// TIA Portal V18 export
// export: Created 2026-06-22T15:41:34.752897Z, ExportSetting WithDefaults, DisplayName Totally Integrated Automation Portal, DisplayVersion V18, DisplayName TIA Portal Openness, DisplayVersion V18, DisplayName TIA Portal Version Control Interface, DisplayVersion V18, DisplayName STEP 7 Professional, DisplayVersion V18, DisplayName STEP 7 Safety, DisplayVersion V18, DisplayName WinCC Professional, DisplayVersion V18
ORGANIZATION_BLOCK "OB30_Encoder_100ms"   // OB30, LAD, CyclicInterrupt
{ S7_Optimized_Access := 'TRUE' }
VERSION : 0.1
// stored: AutoNumber true, IsIECCheckEnabled false, SetENOAutomatically false
   VAR_INPUT
      Initial_Call : Bool;   // Initial call of this OB
      Event_Count : Int;   // Events discarded
   END_VAR
BEGIN

REGION Network 1: Đọc giá trị HSC và tính Delta Count
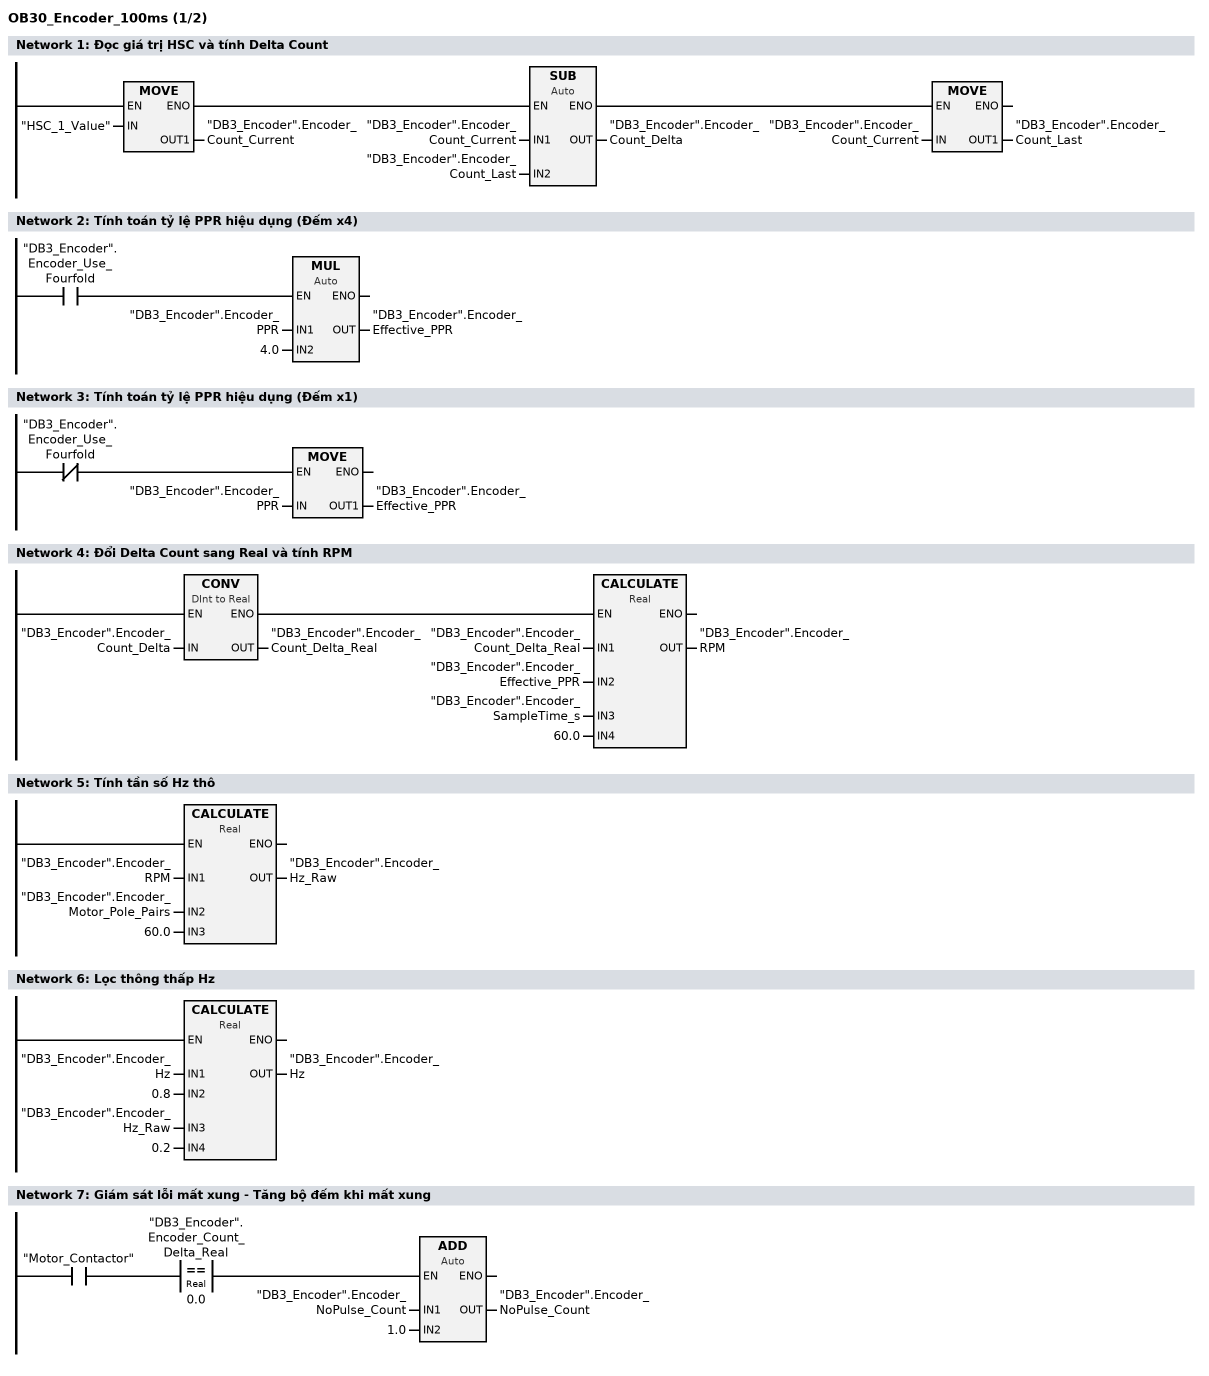
   RUNG wire#powerrail
      { S7_GenerateENO := "TRUE" } Move(in := "HSC_1_Value", out1 => "DB3_Encoder".Encoder_Count_Current)
      { S7_GenerateENO := "TRUE" } Sub(in1 := "DB3_Encoder".Encoder_Count_Current, in2 := "DB3_Encoder".Encoder_Count_Last, out => "DB3_Encoder".Encoder_Count_Delta)
      { S7_GenerateENO := "TRUE" } Move(in := "DB3_Encoder".Encoder_Count_Current, out1 => "DB3_Encoder".Encoder_Count_Last)
   END_RUNG
   // the same network as SCL:
   // ENO of a box is taken as its EN; it also drops when the box reports an error
   "DB3_Encoder".Encoder_Count_Current := "HSC_1_Value";
   "DB3_Encoder".Encoder_Count_Delta := "DB3_Encoder".Encoder_Count_Current - "DB3_Encoder".Encoder_Count_Last;
   "DB3_Encoder".Encoder_Count_Last := "DB3_Encoder".Encoder_Count_Current;
END_REGION

REGION Network 2: Tính toán tỷ lệ PPR hiệu dụng (Đếm x4)
   RUNG wire#powerrail
      Contact( "DB3_Encoder".Encoder_Use_Fourfold )
      { S7_GenerateENO := "TRUE" } Mul(in1 := "DB3_Encoder".Encoder_PPR, in2 := 4.0, out => "DB3_Encoder".Encoder_Effective_PPR)
   END_RUNG
   // the same network as SCL:
   IF "DB3_Encoder".Encoder_Use_Fourfold THEN
       "DB3_Encoder".Encoder_Effective_PPR := "DB3_Encoder".Encoder_PPR * 4.0;
   END_IF;
END_REGION

REGION Network 3: Tính toán tỷ lệ PPR hiệu dụng (Đếm x1)
   RUNG wire#powerrail
      I_Contact( "DB3_Encoder".Encoder_Use_Fourfold )
      { S7_GenerateENO := "TRUE" } Move(in := "DB3_Encoder".Encoder_PPR, out1 => "DB3_Encoder".Encoder_Effective_PPR)
   END_RUNG
   // the same network as SCL:
   IF NOT "DB3_Encoder".Encoder_Use_Fourfold THEN
       "DB3_Encoder".Encoder_Effective_PPR := "DB3_Encoder".Encoder_PPR;
   END_IF;
END_REGION

REGION Network 4: Đổi Delta Count sang Real và tính RPM
   RUNG wire#powerrail
      { S7_Templates := "[SrcType := DInt, DestType := Real]"; S7_GenerateENO := "TRUE" } Convert(in := "DB3_Encoder".Encoder_Count_Delta, out => "DB3_Encoder".Encoder_Count_Delta_Real)
      { S7_Templates := "SrcType := Real"; S7_GenerateENO := "TRUE"; S7_Expression := "(IN1 * IN4) / (IN2 * IN3)" } Calculate(in1 := "DB3_Encoder".Encoder_Count_Delta_Real, in2 := "DB3_Encoder".Encoder_Effective_PPR, in3 := "DB3_Encoder".Encoder_SampleTime_s, in4 := 60.0, out => "DB3_Encoder".Encoder_RPM)
   END_RUNG
   // the same network as SCL:
   // ENO of a box is taken as its EN; it also drops when the box reports an error
   "DB3_Encoder".Encoder_Count_Delta_Real := DINT_TO_REAL("DB3_Encoder".Encoder_Count_Delta);
   "DB3_Encoder".Encoder_RPM := ("DB3_Encoder".Encoder_Count_Delta_Real * 60.0) / ("DB3_Encoder".Encoder_Effective_PPR * "DB3_Encoder".Encoder_SampleTime_s);
END_REGION

REGION Network 5: Tính tần số Hz thô
   RUNG wire#powerrail
      { S7_Templates := "SrcType := Real"; S7_GenerateENO := "TRUE"; S7_Expression := "(IN1 * IN2) / IN3" } Calculate(in1 := "DB3_Encoder".Encoder_RPM, in2 := "DB3_Encoder".Encoder_Motor_Pole_Pairs, in3 := 60.0, out => "DB3_Encoder".Encoder_Hz_Raw)
   END_RUNG
   // the same network as SCL:
   "DB3_Encoder".Encoder_Hz_Raw := ("DB3_Encoder".Encoder_RPM * "DB3_Encoder".Encoder_Motor_Pole_Pairs) / 60.0;
END_REGION

REGION Network 6: Lọc thông thấp Hz
   RUNG wire#powerrail
      { S7_Templates := "SrcType := Real"; S7_GenerateENO := "TRUE"; S7_Expression := "(IN1 * IN2) + (IN3 * IN4)" } Calculate(in1 := "DB3_Encoder".Encoder_Hz, in2 := 0.8, in3 := "DB3_Encoder".Encoder_Hz_Raw, in4 := 0.2, out => "DB3_Encoder".Encoder_Hz)
   END_RUNG
   // the same network as SCL:
   "DB3_Encoder".Encoder_Hz := ("DB3_Encoder".Encoder_Hz * 0.8) + ("DB3_Encoder".Encoder_Hz_Raw * 0.2);
END_REGION

REGION Network 7: Giám sát lỗi mất xung - Tăng bộ đếm khi mất xung
   RUNG wire#powerrail
      Contact( "Motor_Contactor" )
      { S7_Templates := "SrcType := Real" } EQ_Contact(in1 := "DB3_Encoder".Encoder_Count_Delta_Real, in2 := 0.0)
      { S7_GenerateENO := "TRUE" } Add(in1 := "DB3_Encoder".Encoder_NoPulse_Count, in2 := 1.0, out => "DB3_Encoder".Encoder_NoPulse_Count)
   END_RUNG
   // the same network as SCL:
   IF "Motor_Contactor" AND ("DB3_Encoder".Encoder_Count_Delta_Real = 0.0) THEN
       "DB3_Encoder".Encoder_NoPulse_Count := "DB3_Encoder".Encoder_NoPulse_Count + 1.0;
   END_IF;
END_REGION

REGION Network 8: Giám sát lỗi mất xung - Reset bộ đếm khi có xung
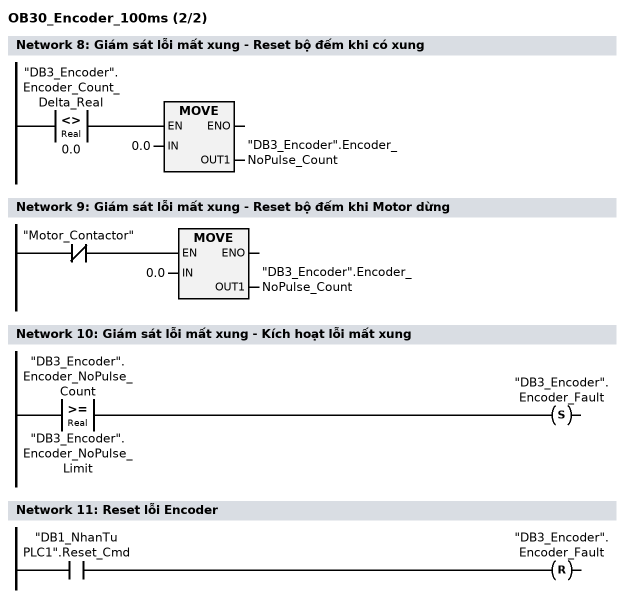
   RUNG wire#powerrail
      { S7_Templates := "SrcType := Real" } NE_Contact(in1 := "DB3_Encoder".Encoder_Count_Delta_Real, in2 := 0.0)
      { S7_GenerateENO := "TRUE" } Move(in := 0.0, out1 => "DB3_Encoder".Encoder_NoPulse_Count)
   END_RUNG
   // the same network as SCL:
   IF "DB3_Encoder".Encoder_Count_Delta_Real <> 0.0 THEN "DB3_Encoder".Encoder_NoPulse_Count := 0.0; END_IF;
END_REGION

REGION Network 9: Giám sát lỗi mất xung - Reset bộ đếm khi Motor dừng
   RUNG wire#powerrail
      I_Contact( "Motor_Contactor" )
      { S7_GenerateENO := "TRUE" } Move(in := 0.0, out1 => "DB3_Encoder".Encoder_NoPulse_Count)
   END_RUNG
   // the same network as SCL:
   IF NOT "Motor_Contactor" THEN "DB3_Encoder".Encoder_NoPulse_Count := 0.0; END_IF;
END_REGION

REGION Network 10: Giám sát lỗi mất xung - Kích hoạt lỗi mất xung
   RUNG wire#powerrail
      { S7_Templates := "SrcType := Real" } GE_Contact(in1 := "DB3_Encoder".Encoder_NoPulse_Count, in2 := "DB3_Encoder".Encoder_NoPulse_Limit)
      S_Coil( "DB3_Encoder".Encoder_Fault )
   END_RUNG
   // the same network as SCL:
   IF "DB3_Encoder".Encoder_NoPulse_Count >= "DB3_Encoder".Encoder_NoPulse_Limit THEN
       "DB3_Encoder".Encoder_Fault := TRUE;
   END_IF;
END_REGION

REGION Network 11: Reset lỗi Encoder
   RUNG wire#powerrail
      Contact( "DB1_NhanTuPLC1".Reset_Cmd )
      R_Coil( "DB3_Encoder".Encoder_Fault )
   END_RUNG
   // the same network as SCL:
   IF "DB1_NhanTuPLC1".Reset_Cmd THEN "DB3_Encoder".Encoder_Fault := FALSE; END_IF;
END_REGION
END_ORGANIZATION_BLOCK
